(* IEC 61131-3 sources: plc_generation_empirical_study/datasets/packages/internal_v0_1_precalibration_20260810/qualification_only/C06_E01_three_part_counter/negative_control, 1 file *)

(* ---- NC1.st ---- *)
FUNCTION_BLOCK C06_E01_three_part_counter
VAR_INPUT
    PartPulse : BOOL;
    Reset : BOOL;
END_VAR
VAR_OUTPUT
    Count : INT;
    Complete : BOOL;
END_VAR
VAR
    PrevPart : BOOL := TRUE;
END_VAR

IF Reset THEN
    Count := 0;
ELSIF PartPulse AND (NOT PrevPart) AND (Count < 3) THEN
    Count := Count + 1;
END_IF;
Complete := Count = 3;
PrevPart := PartPulse;

END_FUNCTION_BLOCK
